INTERFACE I_Button

PROPERTY IsPressed : BOOL
GET
END_GET
END_PROPERTY

END_INTERFACE

(* stored: Version 1.1.0.1, ProductVersion 3.1.4024.12
   Itf I_Button: Id {2e5e0d70-2ab7-4ccb-829a-46e6809f583e}
   Property IsPressed: Id {1c1cc6bd-d448-4fba-bea5-fb716cc6c925}
   Get Get: Id {f7fe1c53-09ba-4c6a-bf43-631a4b753b3b} *)
